(* IEC 61131-3 sources: volt/packages/volt-lsp-iec/test-corpus/CodesysTestProject/Device/Plc Logic/Application/Library Manager/CmpLog, 13 files *)

(* ---- EVTPARAM_CMPLOGADD.dut ---- *)
TYPE EVTPARAM_CMPLOGADD :
STRUCT
	HLOG : RTS_IEC_HANDLE;
	CMPID : UDINT;
	ICLASSID : DINT;
	IERRORID : RTS_IEC_RESULT;
	IINFOID : DINT;
	PSZINFO : POINTER TO STRING;
	PARGLIST : POINTER TO BYTE;
END_STRUCT
END_TYPE

(* ---- LOGOPTIONS.dut ---- *)
TYPE LOGOPTIONS :
STRUCT
	SZNAME : STRING(31);
	BENABLE : DINT;
	UITYPE : UDINT;
	UIFILTER : UDINT;
	IMAXENTRIES : DINT;
	IMAXFILESIZE : DINT;
	IMAXFILES : DINT;
END_STRUCT
END_TYPE

(* ---- EVENTIDS.gvl ---- *)
VAR_GLOBAL
	CMPID_CMPLOG : DWORD := 16#13;
	EVTPARAMID_CMPLOGADD : WORD := 16#1;
	EVTVERSION_CMPLOGADD : WORD := 16#2;
	EVT_LOGADD : DWORD := 16#10001;
END_VAR

(* ---- LOGCLASS.gvl ---- *)
VAR_GLOBAL
	LOG_NONE : UDINT := 16#0;
	LOG_INFO : UDINT := 16#1;
	LOG_WARNING : UDINT := 16#2;
	LOG_ERROR : UDINT := 16#4;
	LOG_EXCEPTION : UDINT := 16#8;
	LOG_DEBUG : UDINT := 16#10;
	LOG_USER_NOTIFY : UDINT := 16#10000;
	LOG_ALL : UDINT := 16#FFFFFFFF;
END_VAR

(* ---- LOGCONSTANTS.gvl ---- *)
VAR_GLOBAL
	STD_LOGGER : RTS_IEC_HANDLE := 0;
	LOG_STD_LOGGER : RTS_IEC_HANDLE := STD_LOGGER;
	LOG_INVALID_HANDLE : RTS_IEC_HANDLE := RTS_INVALID_HANDLE;
END_VAR

(* ---- LOGTYPES.gvl ---- *)
VAR_GLOBAL
	LT_HIGHSPEED : UDINT := 16#1;
	LT_SAFE : UDINT := 16#2;
	LT_NORMAL : UDINT := 16#4;
	LT_TIMESTAMP_RTC : UDINT := 16#10;
	LT_TIMESTAMP_RTC_HIGHRES : UDINT := 16#2000;
	LT_TIMESTAMP_MS : UDINT := 16#20;
	LT_TIMESTAMP_US : UDINT := 16#40;
	LT_TIMESTAMP_NS : UDINT := 16#80;
	LT_NO_DISABLE : UDINT := 16#100;
	LT_DUMP_ASYNC : UDINT := 16#200;
	LT_DUMP_ALWAYS : UDINT := 16#400;
	LT_DUMP_ON_CLOSE : UDINT := 16#800;
	LT_DUMP_ON_REQUEST : UDINT := 16#1000;
	LT_STD : UDINT := (((LT_NORMAL OR LT_TIMESTAMP_RTC) OR LT_NO_DISABLE) OR LT_DUMP_ASYNC);
END_VAR

(* ---- LOGADD.pou ---- *)
FUNCTION LOGADD : RTS_IEC_RESULT
VAR_INPUT
	HLOGGER : RTS_IEC_HANDLE;
	STCMPNAME : STRING(80);
	DICLASSID : DINT;
	DIERRORID : DINT;
	DIINFOID : DINT;
	STINFO : STRING(255);
END_VAR
END_FUNCTION

(* ---- LOGADD2.pou ---- *)
FUNCTION LOGADD2 : RTS_IEC_RESULT
VAR_INPUT
	HLOGGER : RTS_IEC_HANDLE;
	UDICMPID : UDINT;
	UDICLASSID : UDINT;
	UDIERRORID : UDINT;
	UDIINFOID : UDINT;
	PSZINFO : REFERENCE TO STRING;
END_VAR
END_FUNCTION

(* ---- LOGCLOSE.pou ---- *)
FUNCTION LOGCLOSE : RTS_IEC_RESULT
VAR_INPUT
	HLOGGER : RTS_IEC_HANDLE;
END_VAR
END_FUNCTION

(* ---- LOGCOPYINFO.pou ---- *)
FUNCTION LOGCOPYINFO : RTS_IEC_RESULT
VAR_INPUT
	HLOGGER : RTS_IEC_HANDLE;
	PSZINFO : POINTER TO STRING;
	PARGLIST : POINTER TO BYTE;
	PSZSTRING : POINTER TO STRING;
	PDIMAXSTRINGLEN : POINTER TO DINT;
END_VAR
END_FUNCTION

(* ---- LOGCREATE.pou ---- *)
FUNCTION LOGCREATE : RTS_IEC_HANDLE
VAR_INPUT
	POPTIONS : POINTER TO LogOptions;
	PRESULT : POINTER TO RTS_IEC_RESULT;
END_VAR
END_FUNCTION

(* ---- LOGDELETE.pou ---- *)
FUNCTION LOGDELETE : RTS_IEC_RESULT
VAR_INPUT
	HLOGGER : RTS_IEC_HANDLE;
END_VAR
END_FUNCTION

(* ---- LOGOPEN.pou ---- *)
FUNCTION LOGOPEN : RTS_IEC_HANDLE
VAR_INPUT
	PSZNAME : REFERENCE TO STRING;
	PRESULT : POINTER TO RTS_IEC_RESULT;
END_VAR
END_FUNCTION
